// TIA Portal V17 export
// export: Created 2024-09-15T12:30:37.9378246Z, ExportSetting WithDefaults, DisplayName Totally Integrated Automation Portal, DisplayVersion V17, DisplayName TIA Portal Openness, DisplayVersion V17, DisplayName TIA Portal Version Control Interface, DisplayVersion V17, DisplayName STEP 7 Professional, DisplayVersion V17, DisplayName STEP 7 Safety, DisplayVersion V17, DisplayName WinCC Professional, DisplayVersion V17
TYPE "typ_Workpiece_Parameters"
// stored: IsFailsafeCompliant false
   STRUCT
      DoOven : Bool;
      OvenTime : Time;
      DoSaw : Bool;
      SawTime : Time;
   END_STRUCT;
END_TYPE
